// Mitsubishi GX Works2 project: PLC   PLC: FX3G

// global labels: Global1
VAR_GLOBAL
  DuringWorkingDay AT M1 : BOOL;
  StartAmountRasberry AT D1108 : REAL;
  RasberryContainer AT D1100 : REAL;
  StartAmountLemon AT D1110 : REAL;
  LemonContainer AT D1102 : REAL;
  StartAmountStabilizer AT D1114 : REAL;
  StabilizerContainer AT D1106 : REAL;
  StartAmountGummy AT D1112 : REAL;
  GummyContainer AT D1104 : REAL;
  OutPut AT D8282 : INT;
  StartWorkingDay AT X007 : BOOL;
  EmergencySwitch AT X005 : BOOL;
  InventoryIsFinished AT M7 : BOOL;
  EndWorkDay AT M15 : BOOL;
  StartIceCreamMaking AT X001 : BOOL;
  IceCreamMakingTimer AT TC1 : BOOL;
END_VAR
VAR_GLOBAL CONSTANT
  Const50 : INT := 50;
END_VAR
VAR_GLOBAL
  AnalogInput1 AT D8280 : INT;
END_VAR
VAR_GLOBAL CONSTANT
  Const400 : INT := 400;
END_VAR
VAR_GLOBAL
  GumigamType AT D1130 : REAL;
END_VAR
VAR_GLOBAL CONSTANT
  Const6 : REAL := 6.0;
  Const10 : INT := 10;
END_VAR
VAR_GLOBAL
  GumigamPinuk AT M14 : BOOL;
END_VAR
VAR_GLOBAL CONSTANT
  Const_5 : REAL := 5.0;
END_VAR
VAR_GLOBAL
  Pinuk AT M24 : BOOL;
  Packing7Gumigam AT Y004 : BOOL;
  Ragil AT M23 : BOOL;
END_VAR
VAR_GLOBAL CONSTANT
  Const385 : REAL := 385.0;
  Const665 : REAL := 665.0;
  Const210 : REAL := 210.0;
  Const70 : REAL := 70.0;
END_VAR
VAR_GLOBAL
  NotEnoughForPinuk AT M16 : BOOL;
END_VAR
VAR_GLOBAL CONSTANT
  Const280 : REAL := 280.0;
  Const455 : REAL := 455.0;
  Const105 : REAL := 105.0;
  Const_28 : REAL := 28.0;
END_VAR
VAR_GLOBAL
  NotEnoughForRagil AT M17 : BOOL;
  EnoughInventory AT M18 : BOOL;
  RasberryMakingCont AT D1116 : REAL;
END_VAR
VAR_GLOBAL CONSTANT
  Const350 : REAL := 350.0;
END_VAR
VAR_GLOBAL
  LemonMakingCont AT D1118 : REAL;
END_VAR
VAR_GLOBAL CONSTANT
  Const490 : REAL := 490.0;
  Const560 : REAL := 560.0;
  Const700 : REAL := 700.0;
END_VAR
VAR_GLOBAL
  IceCreamMakingCounter AT TC1 : BOOL;
  IceCreamMaking_Timer AT TS1 : BOOL;
  IceCreamInProcess AT Y000 : BOOL;
  IceCreamFreeze AT X002 : BOOL;
  FreezingCont AT D1120 : REAL;
  FreezingTimer AT TC2 : BOOL;
END_VAR
VAR_GLOBAL CONSTANT
  Const80 : INT := 80;
END_VAR
VAR_GLOBAL
  TempUnder10 AT X003 : BOOL;
  IceCreamFreezer AT Y002 : BOOL;
  Freezing_Timer AT TS2 : BOOL;
  MixingCont AT D1122 : REAL;
  MixingRagilTimer AT TC3 : BOOL;
END_VAR
VAR_GLOBAL CONSTANT
  Const30 : INT := 30;
END_VAR
VAR_GLOBAL
  MixingRagil_Timer AT TS3 : BOOL;
  StopTimerRagil AT M20 : BOOL;
  MixingPinukTimer AT TC4 : BOOL;
  MixingPinuk_Timer AT TS4 : BOOL;
  StopTimerPinuk AT M21 : BOOL;
  Blinking AT M22 : BOOL;
  Blinking5Timer AT TC5 : BOOL;
  Blinking5_Timer AT TS5 : BOOL;
  Mix5 AT Y005 : BOOL;
  Blinking6Timer AT TC6 : BOOL;
  Blinking6_Timer AT TS6 : BOOL;
  Mix6 AT Y006 : BOOL;
END_VAR
VAR_GLOBAL CONSTANT
  Const_10 : REAL := 10.0;
END_VAR
VAR_GLOBAL
  StartPacking AT X004 : BOOL;
  PackingGumogam AT X000 : BOOL;
END_VAR
VAR_GLOBAL CONSTANT
  Const7 : INT := 7;
END_VAR
VAR_GLOBAL
  GumigamCounter AT CC1 : BOOL;
  Gumigam_Counter AT CS1 : BOOL;
  CurrentCounterGumigam AT CN1 : INT;
END_VAR
VAR_GLOBAL CONSTANT
  Const1 : INT := 1;
  Const_6 : INT := 6;
END_VAR
VAR_GLOBAL
  StorageCont AT D1124 : REAL;
END_VAR
VAR_GLOBAL CONSTANT
  Const_1 : REAL := 1.0;
  Const40 : REAL := 40.0;
END_VAR
VAR_GLOBAL
  OutputTemp AT D1134 : REAL;
  Start_Freeze AT M70 : BOOL;
END_VAR
VAR_GLOBAL CONSTANT
  Const_400 : REAL := 400.0;
END_VAR
VAR_GLOBAL
  GumigamRagil AT M13 : BOOL;
  WorkingDay AT Y007 : BOOL;
  EndIteration AT M25 : BOOL;
  End_day AT M25 : BOOL;
END_VAR

// task Task_01 (event TRUE, interval 0, priority 31): POU_01

PROGRAM POU_01
VAR
  StartFreeze : BOOL;
END_VAR
(* structured ladder/FBD written out as ST: instructions are called as NAME(EN, inputs, outputs); _pN, _eN, _tN stand for wires *)
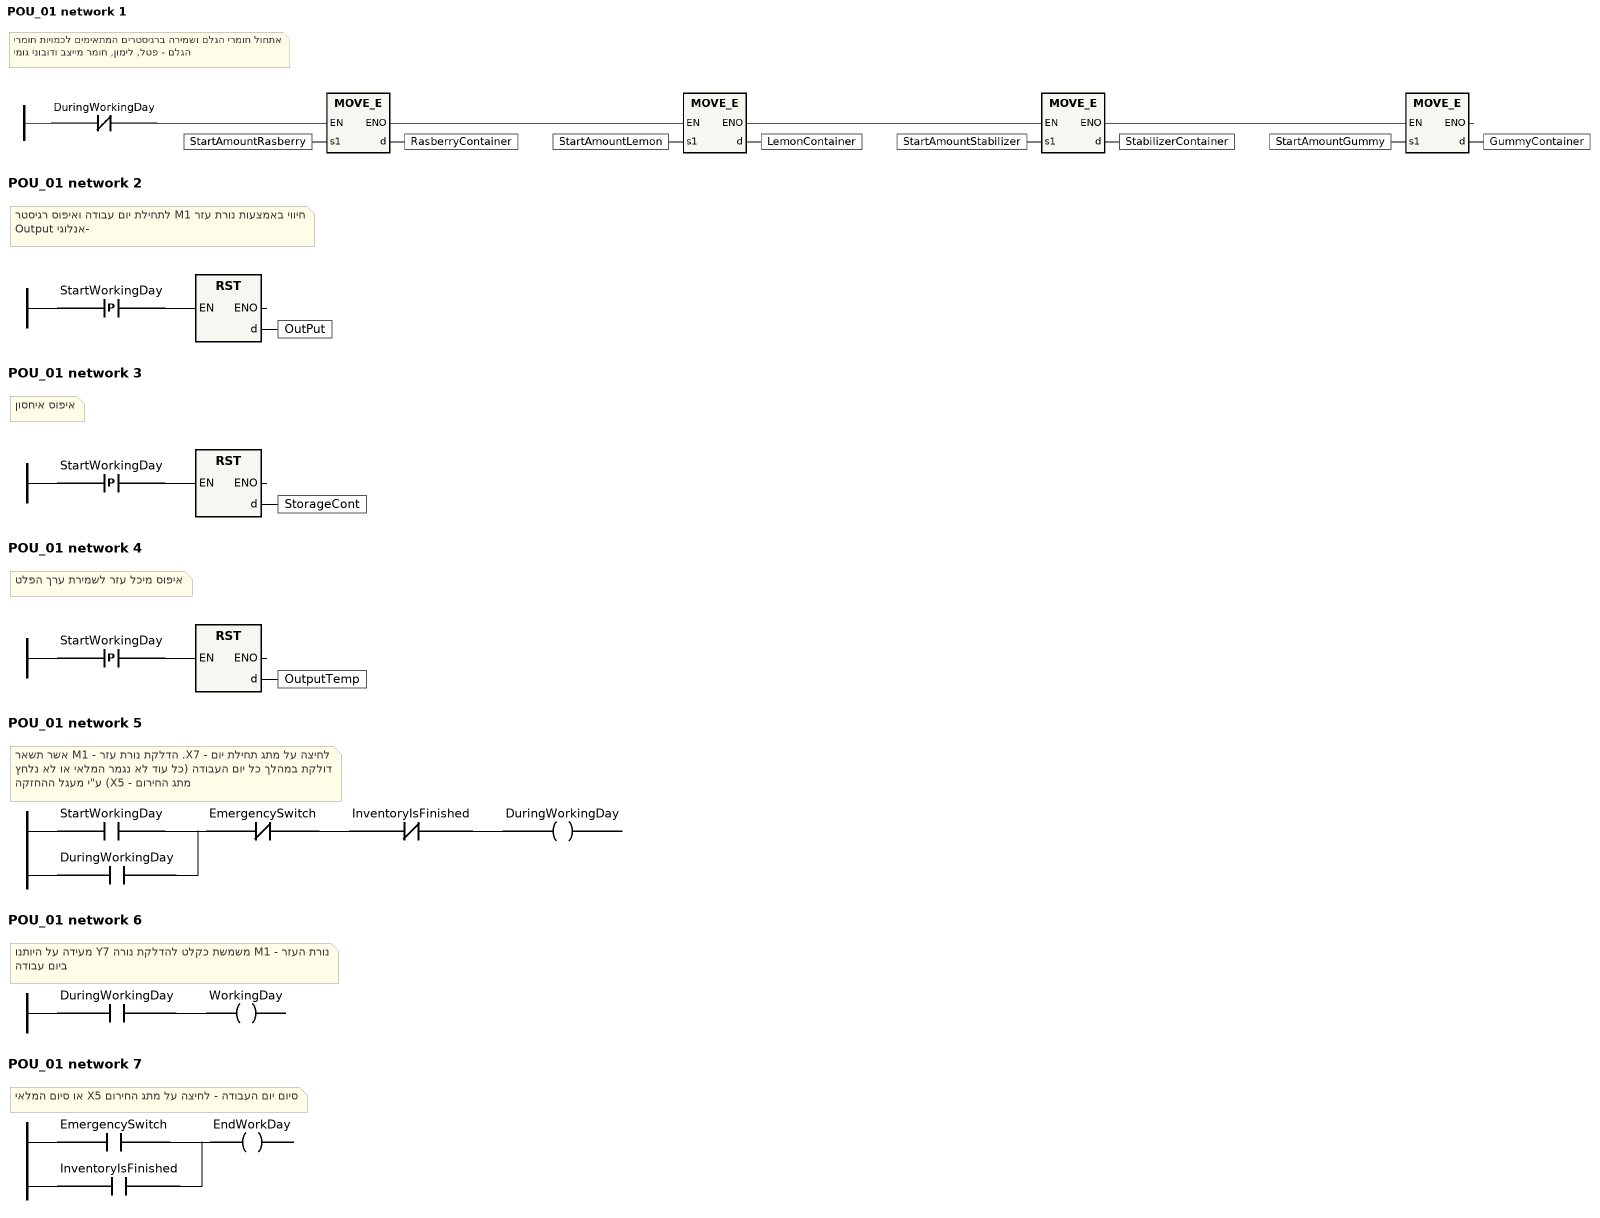
(* network 1 *)
(* אתחול חומרי הגלם ושמירה ברגיסטרים המתאימים לכמויות חומרי הגלם - פטל, לימון, חומר מייצב ודובוני גומי *)
_e1 := MOVE_E(NOT DuringWorkingDay, StartAmountRasberry, RasberryContainer);
_e2 := MOVE_E(_e1, StartAmountLemon, LemonContainer);
_e3 := MOVE_E(_e2, StartAmountStabilizer, StabilizerContainer);
MOVE_E(_e3, StartAmountGummy, GummyContainer);
(* network 2 *)
(* חיווי באמצעות נורת עזר M1 לתחילת יום עבודה ואיפוס רגיסטר Output אנלוגי- *)
RST(LDP(TRUE, StartWorkingDay), OutPut);
(* network 3 *)
(* איפוס איחסון *)
RST(LDP(TRUE, StartWorkingDay), StorageCont);
(* network 4 *)
(* איפוס מיכל עזר לשמירת ערך הפלט *)
RST(LDP(TRUE, StartWorkingDay), OutputTemp);
(* network 5 *)
(* לחיצה על מתג תחילת יום - X7. הדלקת נורת עזר - M1 אשר תשאר דולקת במהלך כל יום העבודה (כל עוד לא נגמר המלאי או לא נלחץ מתג החירום - X5) ע"י מעגל ההחזקה *)
DuringWorkingDay := ((StartWorkingDay OR DuringWorkingDay) AND NOT EmergencySwitch) AND NOT InventoryIsFinished;
(* network 6 *)
(* נורת העזר - M1 משמשת כקלט להדלקת נורה Y7 מעידה על היותנו ביום עבודה *)
WorkingDay := DuringWorkingDay;
(* network 7 *)
(* סיום יום העבודה - לחיצה על מתג החירום X5 או סיום המלאי *)
EndWorkDay := EmergencySwitch OR InventoryIsFinished;
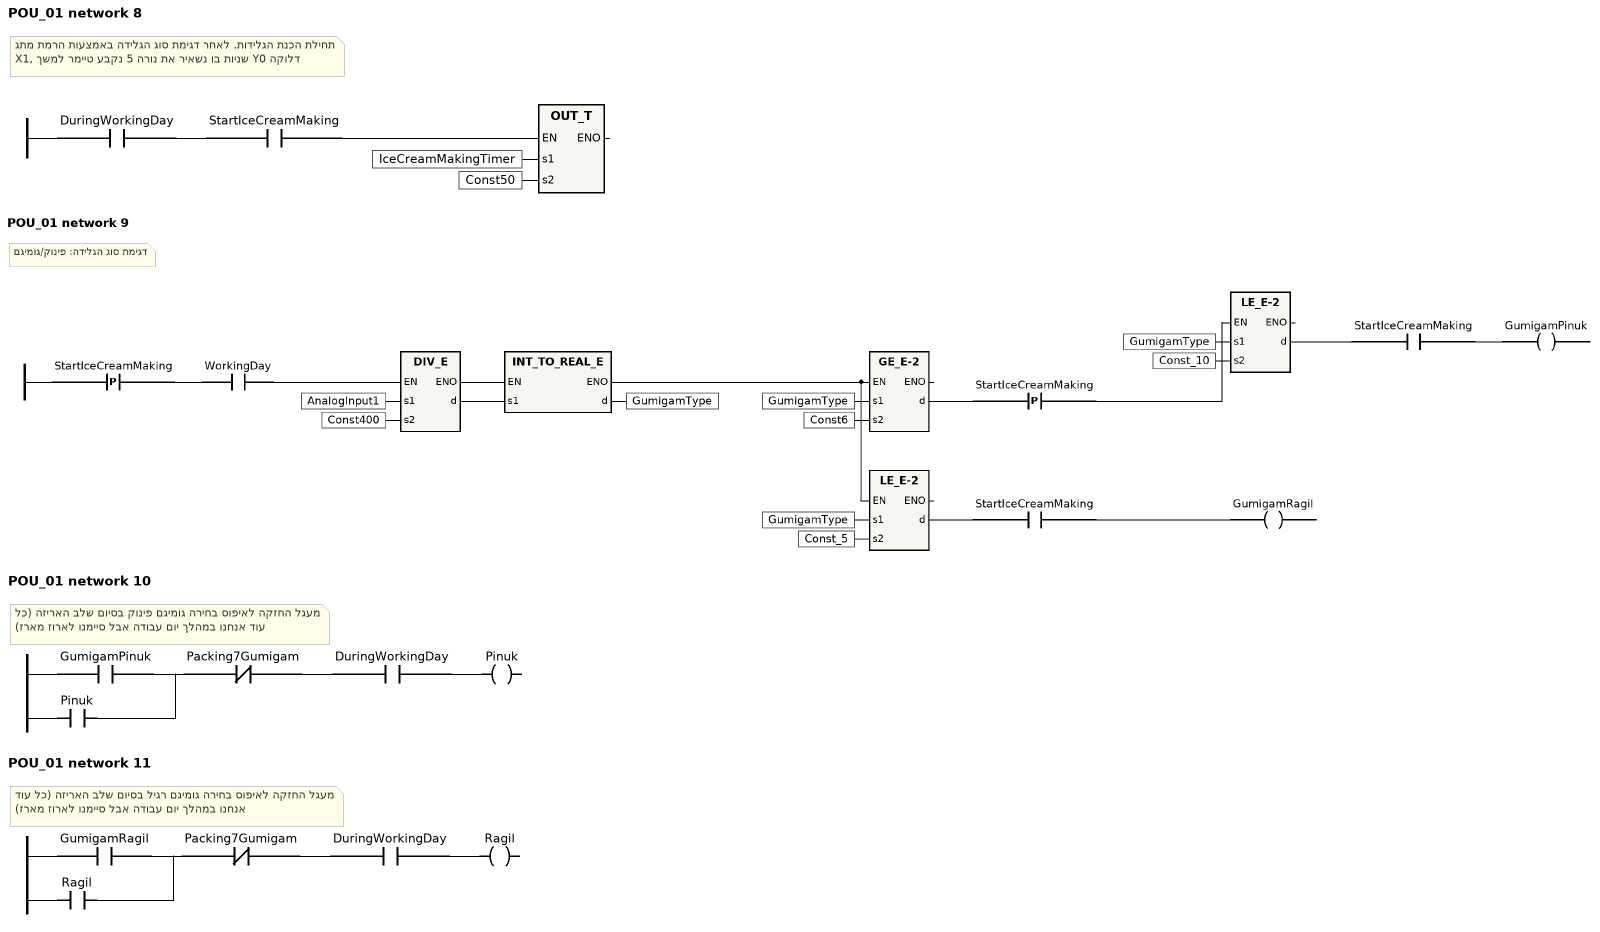
(* network 8 *)
(* תחילת הכנת הגלידות. לאחר דגימת סוג הגלידה באמצעות הרמת מתג X1, נקבע טיימר למשך 5 שניות בו נשאיר את נורה Y0 דלוקה *)
OUT_T(DuringWorkingDay AND StartIceCreamMaking, IceCreamMakingTimer, Const50);
(* network 9 *)
(* דגימת סוג הגלידה: פינוק/גומיגם *)
_e2 := DIV_E(LDP(TRUE, StartIceCreamMaking) AND WorkingDay, AnalogInput1, Const400, _t1);
_e3 := INT_TO_REAL_E(_e2, _t1, GumigamType);
GE_E(_e3, GumigamType, Const6, _t4);
LE_E(_t4 AND LDP(TRUE, StartIceCreamMaking), GumigamType, Const_10, _t5);
GumigamPinuk := _t5 AND StartIceCreamMaking;
LE_E(_e3, GumigamType, Const_5, _t6);
GumigamRagil := _t6 AND StartIceCreamMaking;
(* network 10 *)
(* מעגל החזקה לאיפוס בחירה גומיגם פינוק בסיום שלב האריזה (כל עוד אנחנו במהלך יום עבודה אבל סיימנו לארוז מארז) *)
Pinuk := ((GumigamPinuk OR Pinuk) AND NOT Packing7Gumigam) AND DuringWorkingDay;
(* network 11 *)
(* מעגל החזקה לאיפוס בחירה גומיגם רגיל בסיום שלב האריזה (כל עוד אנחנו במהלך יום עבודה אבל סיימנו לארוז מארז) *)
Ragil := ((GumigamRagil OR Ragil) AND NOT Packing7Gumigam) AND DuringWorkingDay;
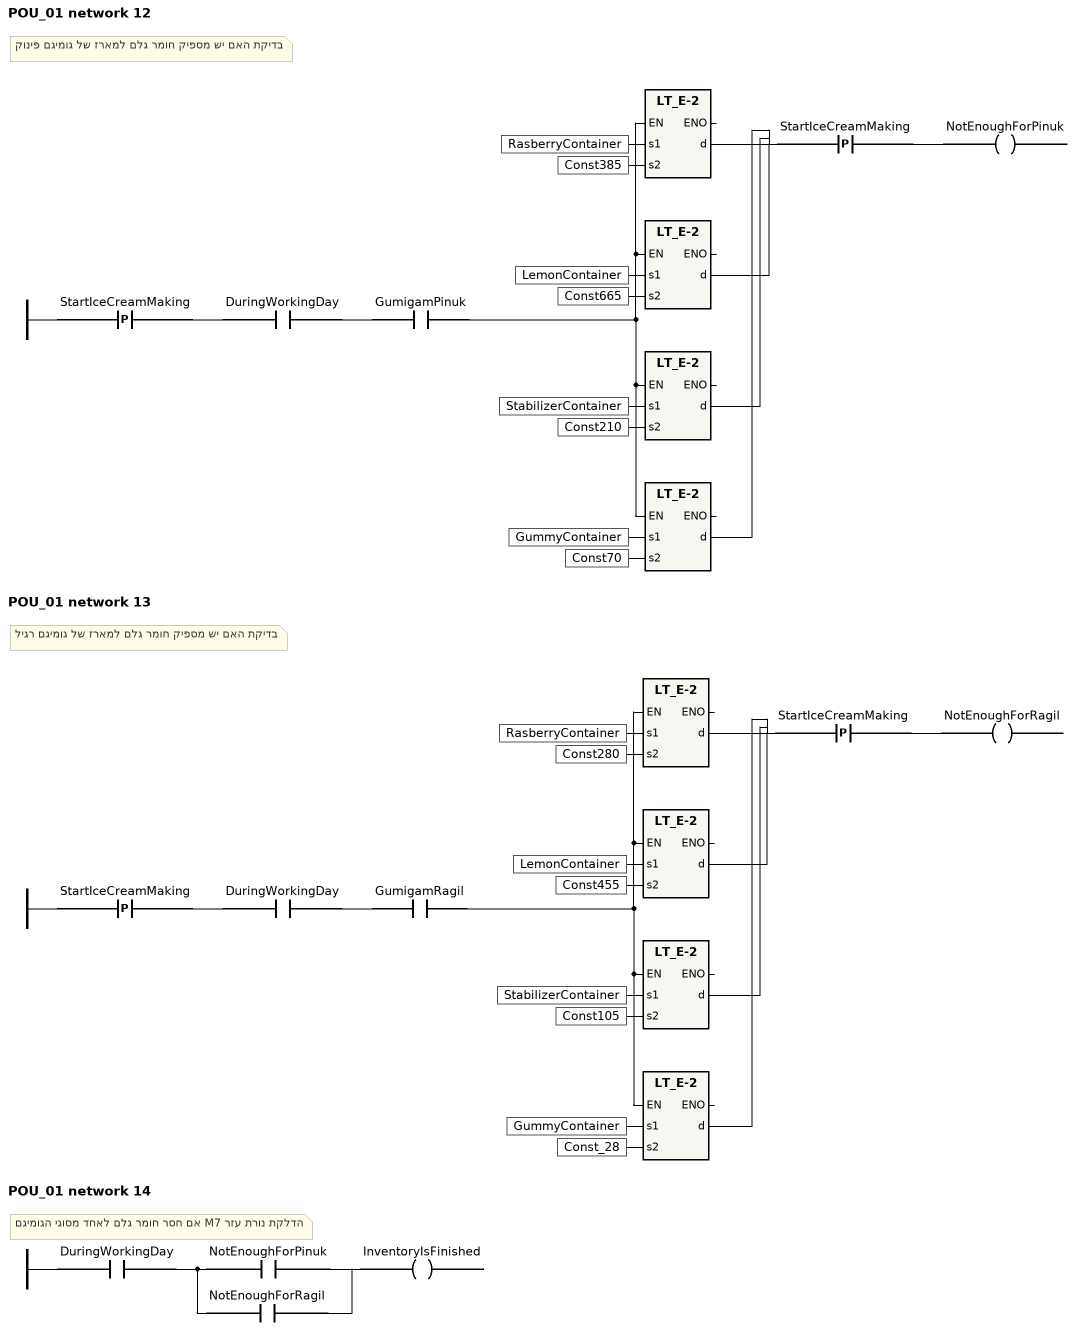
(* network 12 *)
(* בדיקת האם יש מספיק חומר גלם למארז של גומיגם פינוק *)
_p1 := LDP(TRUE, StartIceCreamMaking) AND DuringWorkingDay AND GumigamPinuk;
LT_E(_p1, RasberryContainer, Const385, _t2);
LT_E(_p1, LemonContainer, Const665, _t3);
LT_E(_p1, StabilizerContainer, Const210, _t4);
LT_E(_p1, GummyContainer, Const70, _t5);
NotEnoughForPinuk := (_t2 OR _t3 OR _t4 OR _t5) AND LDP(TRUE, StartIceCreamMaking);
(* network 13 *)
(* בדיקת האם יש מספיק חומר גלם למארז של גומיגם רגיל *)
_p1 := LDP(TRUE, StartIceCreamMaking) AND DuringWorkingDay AND GumigamRagil;
LT_E(_p1, RasberryContainer, Const280, _t2);
LT_E(_p1, LemonContainer, Const455, _t3);
LT_E(_p1, StabilizerContainer, Const105, _t4);
LT_E(_p1, GummyContainer, Const_28, _t5);
NotEnoughForRagil := (_t2 OR _t3 OR _t4 OR _t5) AND LDP(TRUE, StartIceCreamMaking);
(* network 14 *)
(* הדלקת נורת עזר M7 אם חסר חומר גלם לאחד מסוגי הגומיגם *)
InventoryIsFinished := (DuringWorkingDay AND NotEnoughForPinuk) OR (DuringWorkingDay AND NotEnoughForRagil);
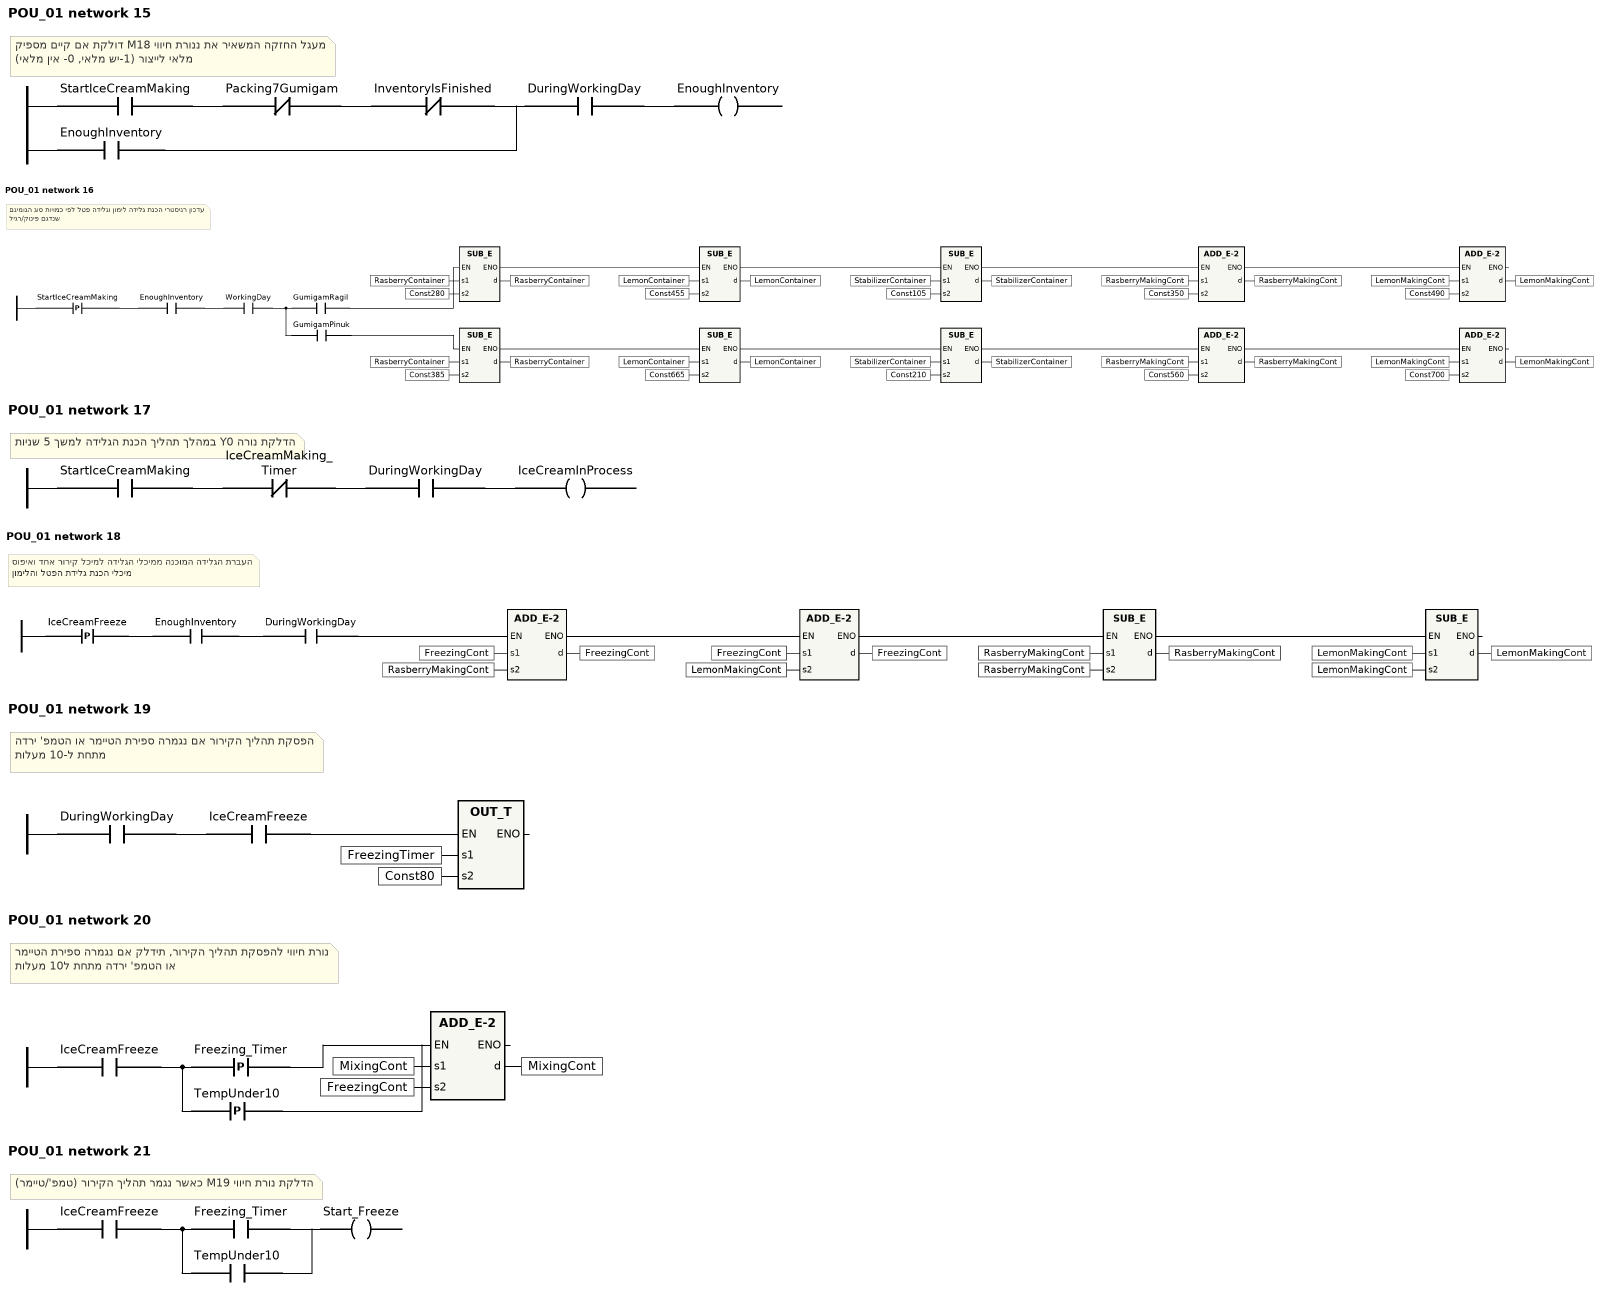
(* network 15 *)
(* מעגל החזקה המשאיר את ננורת חיווי M18 דולקת אם קיים מספיק מלאי לייצור (1-יש מלאי, 0- אין מלאי) *)
EnoughInventory := ((StartIceCreamMaking AND NOT Packing7Gumigam AND NOT InventoryIsFinished) OR EnoughInventory) AND DuringWorkingDay;
(* network 16 *)
(* עדכון רגיסטרי הכנת גלידה לימון וגלידה פטל לפי כמויות סוג הגומיגם שנדגם פינוק/רגיל *)
_p1 := LDP(TRUE, StartIceCreamMaking) AND EnoughInventory AND WorkingDay;
_e2 := SUB_E(_p1 AND GumigamRagil, RasberryContainer, Const280, RasberryContainer);
_e3 := SUB_E(_e2, LemonContainer, Const455, LemonContainer);
_e4 := SUB_E(_e3, StabilizerContainer, Const105, StabilizerContainer);
_e5 := ADD_E(_e4, RasberryMakingCont, Const350, RasberryMakingCont);
ADD_E(_e5, LemonMakingCont, Const490, LemonMakingCont);
_e6 := SUB_E(_p1 AND GumigamPinuk, RasberryContainer, Const385, RasberryContainer);
_e7 := SUB_E(_e6, LemonContainer, Const665, LemonContainer);
_e8 := SUB_E(_e7, StabilizerContainer, Const210, StabilizerContainer);
_e9 := ADD_E(_e8, RasberryMakingCont, Const560, RasberryMakingCont);
ADD_E(_e9, LemonMakingCont, Const700, LemonMakingCont);
(* network 17 *)
(* הדלקת נורה Y0 במהלך תהליך הכנת הגלידה למשך 5 שניות *)
IceCreamInProcess := StartIceCreamMaking AND NOT IceCreamMaking_Timer AND DuringWorkingDay;
(* network 18 *)
(* העברת הגלידה המוכנה ממיכלי הגלידה למיכל קירור אחד ואיפוס מיכלי הכנת גלידת הפטל והלימון *)
_e1 := ADD_E(LDP(TRUE, IceCreamFreeze) AND EnoughInventory AND DuringWorkingDay, FreezingCont, RasberryMakingCont, FreezingCont);
_e2 := ADD_E(_e1, FreezingCont, LemonMakingCont, FreezingCont);
_e3 := SUB_E(_e2, RasberryMakingCont, RasberryMakingCont, RasberryMakingCont);
SUB_E(_e3, LemonMakingCont, LemonMakingCont, LemonMakingCont);
(* network 19 *)
(* הפסקת תהליך הקירור אם נגמרה ספירת הטיימר או הטמפ' ירדה מתחת ל-10 מעלות *)
OUT_T(DuringWorkingDay AND IceCreamFreeze, FreezingTimer, Const80);
(* network 20 *)
(* נורת חיווי להפסקת תהליך הקירור, תידלק אם נגמרה ספירת הטיימר או הטמפ' ירדה מתחת ל10 מעלות *)
ADD_E((IceCreamFreeze AND LDP(TRUE, Freezing_Timer)) OR (IceCreamFreeze AND LDP(TRUE, TempUnder10)), MixingCont, FreezingCont, MixingCont);
(* network 21 *)
(* הדלקת נורת חיווי M19 כאשר נגמר תהליך הקירור (טמפ'/טיימר) *)
Start_Freeze := (IceCreamFreeze AND Freezing_Timer) OR (IceCreamFreeze AND TempUnder10);
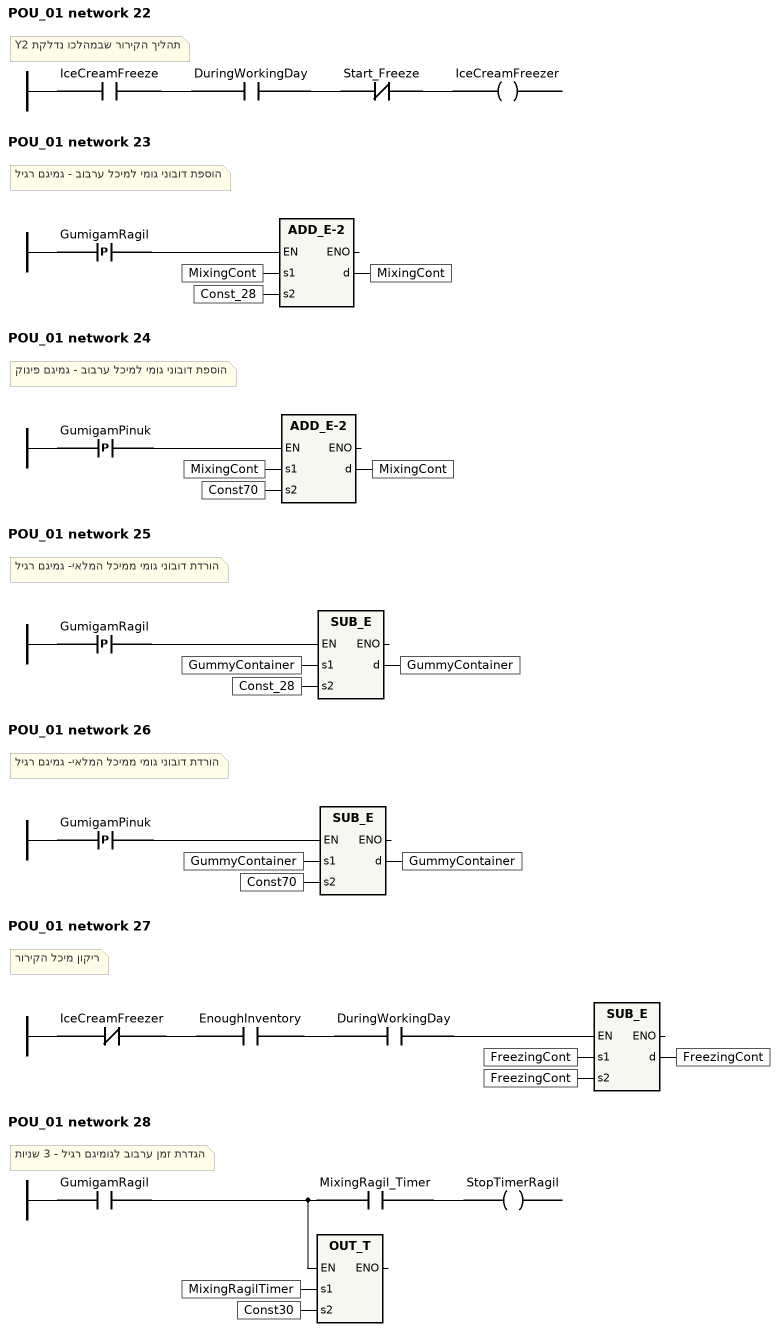
(* network 22 *)
(* תהליך הקירור שבמהלכו נדלקת Y2 *)
IceCreamFreezer := IceCreamFreeze AND DuringWorkingDay AND NOT Start_Freeze;
(* network 23 *)
(* הוספת דובוני גומי למיכל ערבוב - גמיגם רגיל *)
ADD_E(LDP(TRUE, GumigamRagil), MixingCont, Const_28, MixingCont);
(* network 24 *)
(* הוספת דובוני גומי למיכל ערבוב - גמיגם פינוק *)
ADD_E(LDP(TRUE, GumigamPinuk), MixingCont, Const70, MixingCont);
(* network 25 *)
(* הורדת דובוני גומי ממיכל המלאי- גמיגם רגיל *)
SUB_E(LDP(TRUE, GumigamRagil), GummyContainer, Const_28, GummyContainer);
(* network 26 *)
(* הורדת דובוני גומי ממיכל המלאי- גמיגם רגיל *)
SUB_E(LDP(TRUE, GumigamPinuk), GummyContainer, Const70, GummyContainer);
(* network 27 *)
(* ריקון מיכל הקירור *)
SUB_E(NOT IceCreamFreezer AND EnoughInventory AND DuringWorkingDay, FreezingCont, FreezingCont, FreezingCont);
(* network 28 *)
(* הגדרת זמן ערבוב לגומיגם רגיל - 3 שניות *)
StopTimerRagil := GumigamRagil AND MixingRagil_Timer;
OUT_T(GumigamRagil, MixingRagilTimer, Const30);
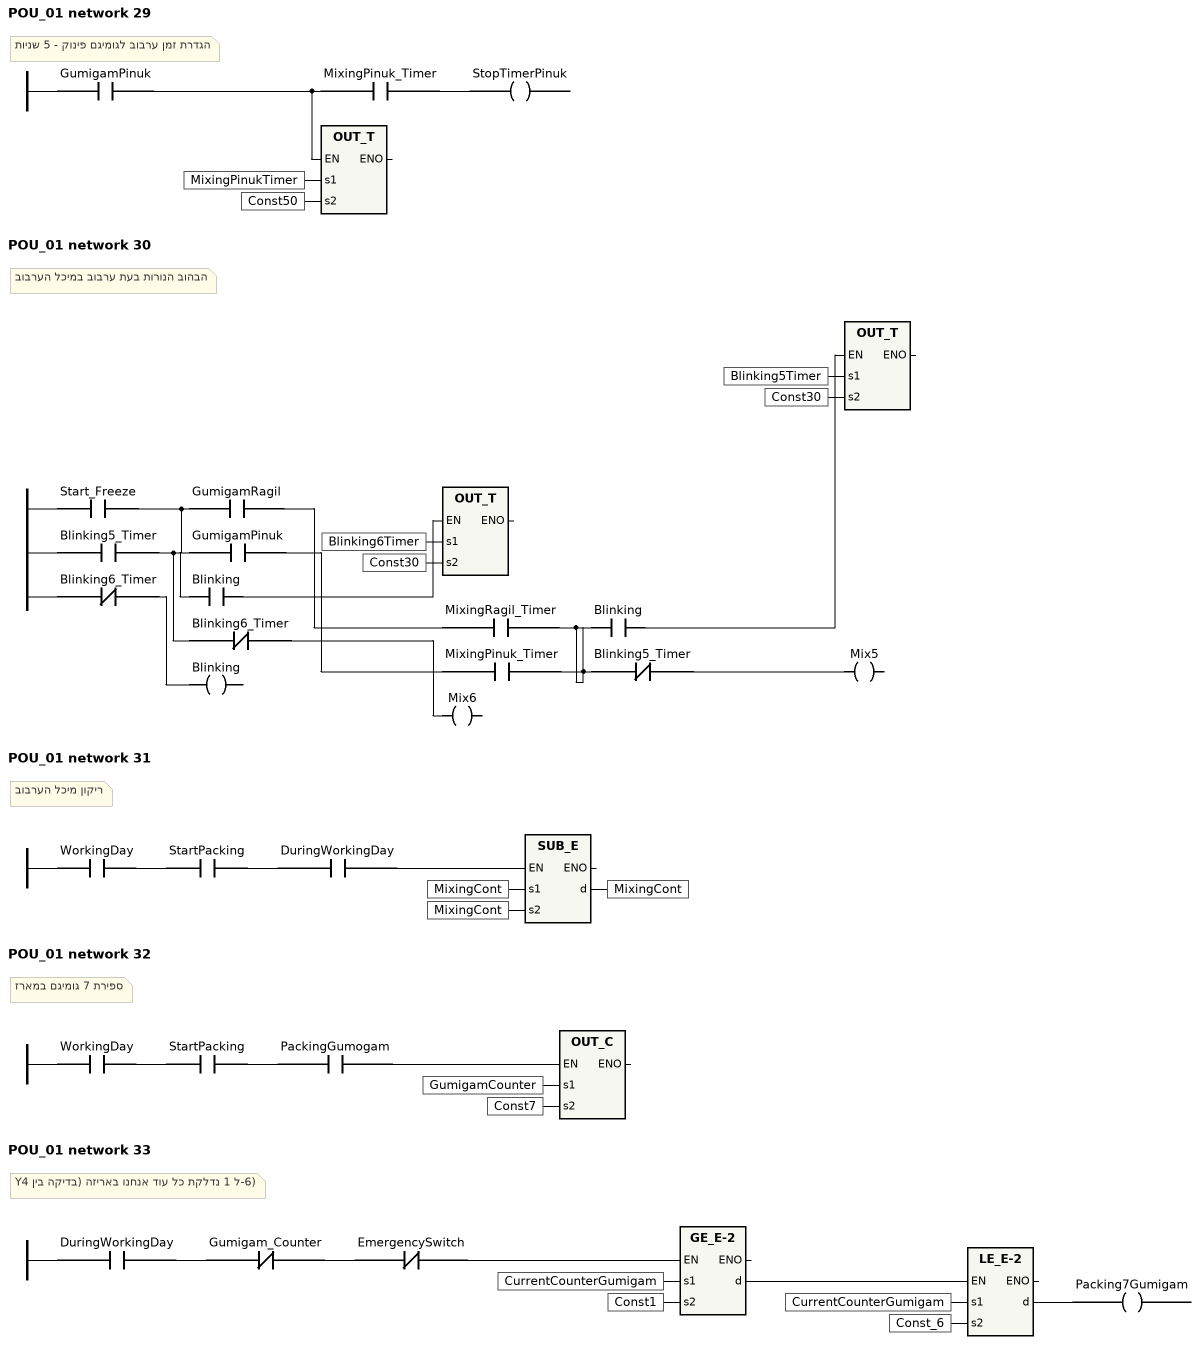
(* network 29 *)
(* הגדרת זמן ערבוב לגומיגם פינוק - 5 שניות *)
StopTimerPinuk := GumigamPinuk AND MixingPinuk_Timer;
OUT_T(GumigamPinuk, MixingPinukTimer, Const50);
(* network 30 *)
(* הבהוב הנורות בעת ערבוב במיכל הערבוב *)
_p1 := (Start_Freeze AND GumigamRagil AND MixingRagil_Timer) OR (Start_Freeze AND GumigamPinuk AND MixingPinuk_Timer);
OUT_T(_p1 AND Blinking, Blinking5Timer, Const30);
Mix5 := _p1 AND NOT Blinking5_Timer;
OUT_T(Blinking5_Timer AND Blinking, Blinking6Timer, Const30);
Mix6 := Blinking5_Timer AND NOT Blinking6_Timer;
Blinking := NOT Blinking6_Timer;
(* network 31 *)
(* ריקון מיכל הערבוב *)
SUB_E(WorkingDay AND StartPacking AND DuringWorkingDay, MixingCont, MixingCont, MixingCont);
(* network 32 *)
(* ספירת 7 גומיגם במארז *)
OUT_C(WorkingDay AND StartPacking AND PackingGumogam, GumigamCounter, Const7);
(* network 33 *)
(* Y4 נדלקת כל עוד אנחנו באריזה (בדיקה בין 1 ל-6) *)
GE_E(DuringWorkingDay AND NOT Gumigam_Counter AND NOT EmergencySwitch, CurrentCounterGumigam, Const1, _t1);
LE_E(_t1, CurrentCounterGumigam, Const_6, _t2);
Packing7Gumigam := _t2;
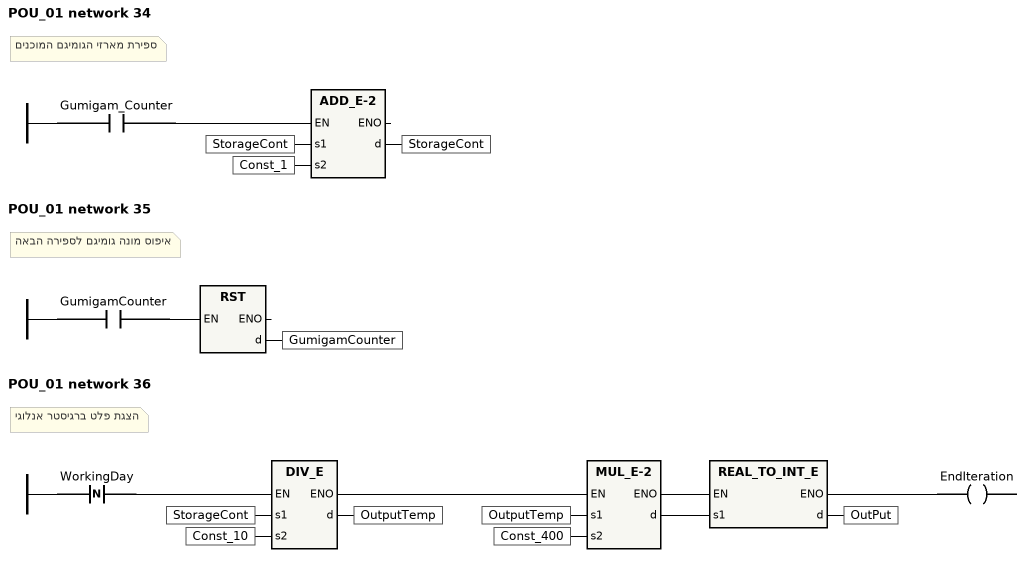
(* network 34 *)
(* ספירת מארזי הגומיגם המוכנים *)
ADD_E(Gumigam_Counter, StorageCont, Const_1, StorageCont);
(* network 35 *)
(* איפוס מונה גומיגם לספירה הבאה *)
RST(GumigamCounter, GumigamCounter);
(* network 36 *)
(* הצגת פלט ברגיסטר אנלוגי *)
_e1 := DIV_E(LDF(TRUE, WorkingDay), StorageCont, Const_10, OutputTemp);
_e3 := MUL_E(_e1, OutputTemp, Const_400, _t2);
_e4 := REAL_TO_INT_E(_e3, _t2, OutPut);
EndIteration := _e4;
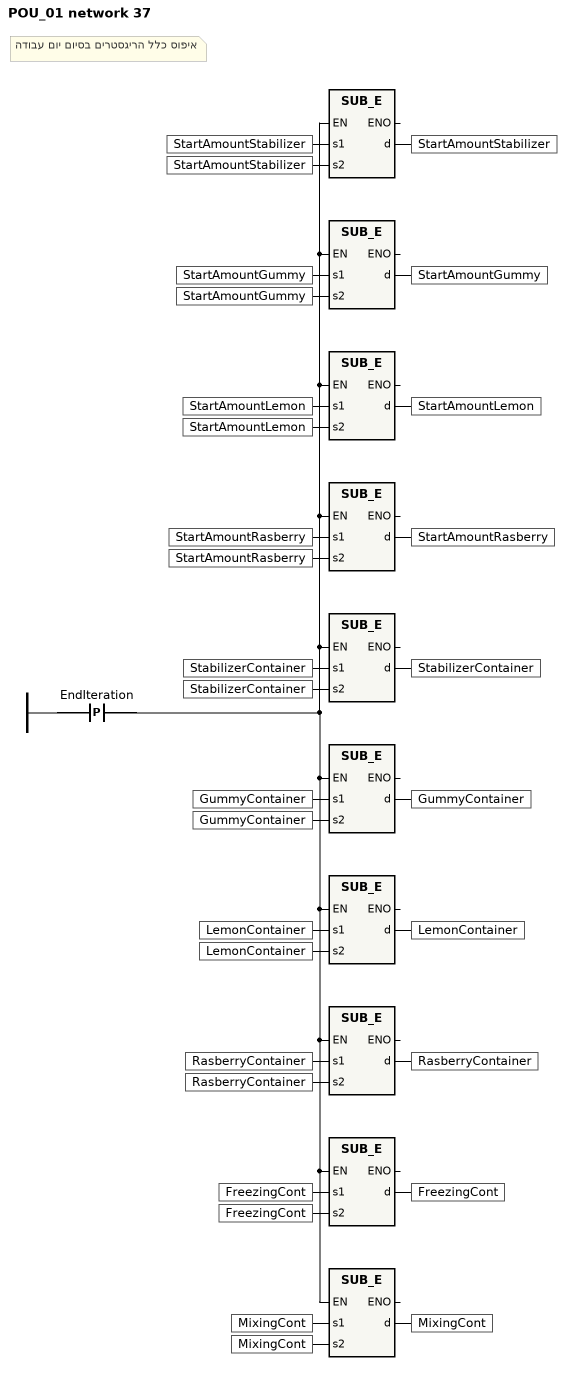
(* network 37 *)
(* איפוס כלל הריגסטרים בסיום יום עבודה *)
_p1 := LDP(TRUE, EndIteration);
SUB_E(_p1, StartAmountStabilizer, StartAmountStabilizer, StartAmountStabilizer);
SUB_E(_p1, StartAmountGummy, StartAmountGummy, StartAmountGummy);
SUB_E(_p1, StartAmountLemon, StartAmountLemon, StartAmountLemon);
SUB_E(_p1, StartAmountRasberry, StartAmountRasberry, StartAmountRasberry);
SUB_E(_p1, StabilizerContainer, StabilizerContainer, StabilizerContainer);
SUB_E(_p1, GummyContainer, GummyContainer, GummyContainer);
SUB_E(_p1, LemonContainer, LemonContainer, LemonContainer);
SUB_E(_p1, RasberryContainer, RasberryContainer, RasberryContainer);
SUB_E(_p1, FreezingCont, FreezingCont, FreezingCont);
SUB_E(_p1, MixingCont, MixingCont, MixingCont);
END_PROGRAM
